// this class implements the main state machine, witch controls the olperations in automatic mode
FUNCTION_BLOCK mainStateMachine_t
VAR_INPUT
	IOExpantionHandler : POINTER TO IOExpantionHandler_t := NULL;
END_VAR
VAR_OUTPUT
END_VAR
VAR
	(* main envorment variables *)	

	isStateMachineOn : BOOL := FALSE; // is stae machine running or not
	stateMachineState : mainStateMachineStatus_t := mainStateMachineStatus_t.IDLE;
	
	startSceduled : BOOL := FALSE; // if true, the "api" has requested the start of the state machine
	stopSceduled : BOOL := FALSE; // if true, the "api" has requzested a stop of the state machine
	
	isStateMachinePaused : BOOL := FALSE;
	
	
	(* RotateTable variables *)	
	
	RotateTable_firstRun : BOOL := TRUE; 		// true when RotateTable is run the first time
	RotateTable_initialState : BOOL := FALSE;	// is the initial state of the TurnTable pos reached sensor
	RotateTable_waitOnRechingPos : TON;
	
	
	(* GripperDown variables *)

	GripperDown_waitUntilNextStep : TON;	
	
	
	(* GripperClose variables *)

	GripperClose_waitUntilNextStep : TON;	
	
	
	(* GripperUp variables *)

	GripperUp_waitUntilNextStep : TON;	
	
	(* GripperDownLeft variables *)

	GripperDownLeft_waitUntilNextStep : TON;	
	
	
	(* GripperOpen variables *)

	GripperOpen_waitUntilNextStep : TON;
	
	(* GripperUpLeft variables *)

	GripperUpLeft_waitUntilNextStep : TON;
	
	(* Y10Out variables *)

	Y10Out_waitUntilNextStep : TON;
	
	
	(* Y10Back variables *)

	Y10Back_waitUntilNextStep : TON;
END_VAR

METHOD PRIVATE convayorbeltStop : BOOL
VAR_INPUT
END_VAR
IOExpantionHandler^.setActor(actorID := actorID_t.ACTOR_Y2_OUT, false);
IOExpantionHandler^.setActor(actorID := actorID_t.ACTOR_Y3_OUT, false);
InputOutput.ConvaorbeltMotorRun := FALSE;

THIS^.stateMachineState := mainStateMachineStatus_t.IDLE; // move on to next step
END_METHOD

METHOD PRIVATE conveyorbeltStart : BOOL
VAR_INPUT
END_VAR
InputOutput.ConvaorbeltMotorRun := TRUE;

IF IOExpantionHandler^.getSensorStatus(sensorID := sensorID_t.EXPANTION_SENSOR_B7_ENTRANCE_CONVAYORBELT) = TRUE THEN
	THIS^.stateMachineState := mainStateMachineStatus_t.Y10_BACK; // move on to next step
END_IF
END_METHOD

METHOD getIsStateMachineON : BOOL
VAR_INPUT
END_VAR
getIsStateMachineON := THIS^.isStateMachineOn;

return;
END_METHOD

METHOD getStateMachineStatus : string
VAR_INPUT
END_VAR
getStateMachineStatus := to_string(THIS^.stateMachineState);

return;
END_METHOD

METHOD PRIVATE GripperClose : BOOL
VAR_INPUT
END_VAR
GripperClose_waitUntilNextStep.PT := T#500MS;

// reset TON
IF GripperClose_waitUntilNextStep.IN = TRUE AND GripperClose_waitUntilNextStep.Q = TRUE THEN
	GripperClose_waitUntilNextStep.IN := FALSE;
	GripperClose_waitUntilNextStep();
END_IF

GripperClose_waitUntilNextStep.IN := TRUE;
GripperClose_waitUntilNextStep();

IF GripperClose_waitUntilNextStep.Q = TRUE THEN
	GripperClose_waitUntilNextStep.IN := FALSE;
	GripperClose_waitUntilNextStep();
	
	IOExpantionHandler^.setActor(actorID := actorID_t.ACTOR_GRIPPER_OPEN_CLOSE, TRUE);
	
	THIS^.stateMachineState := mainStateMachineStatus_t.GRIPPER_UP; // move on to next step
END_IF
END_METHOD

METHOD PRIVATE GripperDown : BOOL
VAR_INPUT
END_VAR
IF GripperDown_waitUntilNextStep.IN = TRUE AND GripperDown_waitUntilNextStep.Q = TRUE THEN
	GripperDown_waitUntilNextStep.IN := FALSE;
	GripperDown_waitUntilNextStep();
END_IF

THIS^.IOExpantionHandler^.setActor(actorID_t.ACTOR_GRIPPER_RIGHT_LEFT, FALSE);

IF IOExpantionHandler^.getSensorStatus(sensorID := sensorID_t.SENSOR_B17_GRIPPER_RIGHT) = FALSE THEN
	// wait (gripper is not on the right)
	RETURN;
END_IF

// configure GripperDown_waitUntilNextStep
GripperDown_waitUntilNextStep.PT := T#500ms;

GripperDown_waitUntilNextStep.IN := TRUE;
GripperDown_waitUntilNextStep();


IOExpantionHandler^.setActor(actorID := actorID_t.ACTOR_GRIPPER_UP_DOWN, TRUE);

IF GripperDown_waitUntilNextStep.Q = FALSE THEN
	RETURN;
END_IF

GripperDown_waitUntilNextStep.IN := FALSE;
GripperDown_waitUntilNextStep();

THIS^.stateMachineState := mainStateMachineStatus_t.GRIPPER_CLOSE; // move on to next step
END_METHOD

METHOD PRIVATE GripperDownLeft : BOOL
VAR_INPUT
END_VAR
GripperDownLeft_waitUntilNextStep.PT := T#1S;

IF GripperDownLeft_waitUntilNextStep.IN = TRUE AND GripperDownLeft_waitUntilNextStep.Q = TRUE THEN
	GripperDownLeft_waitUntilNextStep.IN := FALSE;
	GripperDownLeft_waitUntilNextStep();
END_IF

GripperDownLeft_waitUntilNextStep.IN := TRUE;
GripperDownLeft_waitUntilNextStep();

IOExpantionHandler^.setActor(actorID := actorID_t.ACTOR_GRIPPER_UP_DOWN, TRUE);

IF GripperDownLeft_waitUntilNextStep.Q = TRUE THEN
	GripperDownLeft_waitUntilNextStep.IN := FALSE;
	GripperDownLeft_waitUntilNextStep();	
	
	THIS^.stateMachineState := mainStateMachineStatus_t.GRIPPER_OPEN; // move on to next step
END_IF
END_METHOD

METHOD PRIVATE GripperLeft : BOOL
VAR_INPUT
END_VAR

IOExpantionHandler^.setActor(actorID := actorID_t.ACTOR_GRIPPER_RIGHT_LEFT, true);

IF IOExpantionHandler^.getSensorStatus(sensorID := sensorID_t.SENSOR_B16_GRIPPER_LEFT) = TRUE THEN
	THIS^.stateMachineState := mainStateMachineStatus_t.GRIPPER_DOWN_LEFT; // move on to next step
END_IF
END_METHOD

METHOD PRIVATE GripperOpen : BOOL
VAR_INPUT
END_VAR
GripperOpen_waitUntilNextStep.PT := T#200MS;

IF GripperOpen_waitUntilNextStep.IN = TRUE AND GripperOpen_waitUntilNextStep.Q = TRUE THEN
	GripperOpen_waitUntilNextStep.IN := FALSE;
	GripperOpen_waitUntilNextStep();
END_IF

GripperOpen_waitUntilNextStep.IN := TRUE;
GripperOpen_waitUntilNextStep();

IOExpantionHandler^.setActor(actorID := actorID_t.ACTOR_GRIPPER_OPEN_CLOSE, FALSE);

IF GripperOpen_waitUntilNextStep.Q = TRUE THEN
	GripperOpen_waitUntilNextStep.IN := FALSE;
	GripperOpen_waitUntilNextStep();

	THIS^.stateMachineState := mainStateMachineStatus_t.GRIPPER_UP_LEFT; // move on to next step
END_IF
END_METHOD

METHOD PRIVATE GripperRight : BOOL
VAR_INPUT
END_VAR
END_METHOD

METHOD PRIVATE GripperUp : BOOL
VAR_INPUT
END_VAR
VAR 
	
END_VAR
GripperUp_waitUntilNextStep.PT := T#500MS;

IF GripperUp_waitUntilNextStep.IN = TRUE AND GripperUp_waitUntilNextStep.Q = TRUE THEN
	GripperUp_waitUntilNextStep.IN := FALSE;
	GripperUp_waitUntilNextStep();
END_IF

GripperUp_waitUntilNextStep.IN := TRUE;
GripperUp_waitUntilNextStep();


IF GripperUp_waitUntilNextStep.Q = TRUE THEN
	IOExpantionHandler^.setActor(actorID := actorID_t.ACTOR_GRIPPER_UP_DOWN, FALSE);
	THIS^.stateMachineState := mainStateMachineStatus_t.GRIPPER_LEFT; // move on to next step
END_IF
END_METHOD

METHOD PRIVATE GripperUpLeft : BOOL
VAR_INPUT
END_VAR
GripperUpLeft_waitUntilNextStep.PT := T#500MS;

IF GripperUpLeft_waitUntilNextStep.IN = TRUE AND GripperUpLeft_waitUntilNextStep.Q = TRUE THEN
	GripperUpLeft_waitUntilNextStep.IN := FALSE;
	GripperUpLeft_waitUntilNextStep();
END_IF


IOExpantionHandler^.setActor(actorID := actorID_t.ACTOR_GRIPPER_UP_DOWN, FALSE);

GripperUpLeft_waitUntilNextStep.IN := TRUE;
GripperUpLeft_waitUntilNextStep();	

IF GripperUpLeft_waitUntilNextStep.Q = TRUE THEN
	GripperUpLeft_waitUntilNextStep.IN := FALSE;
	GripperUpLeft_waitUntilNextStep();	

	IF IOExpantionHandler^.getSensorStatus(sensorID := sensorID_t.EXPANTION_SENSOR_B7_ENTRANCE_CONVAYORBELT) = TRUE THEN
		THIS^.stateMachineState := mainStateMachineStatus_t.CONVAYORBELT_START; // move on to next step
	ELSE 
		THIS^.stateMachineState := mainStateMachineStatus_t.Y10_OUT; // move on to next step
	END_IF;
END_IF
END_METHOD

// if this function is called, the statemachine pauses its execution and stores its state, all movement will be paused or will wait until all movment is paused. A mutch "safer" alternative to reset()
METHOD pause : BOOL
VAR_INPUT
	isPaused : BOOL := TRUE;	
END_VAR
IF THIS^.isStateMachineOn = FALSE THEN
	pause := FALSE;
	RETURN;
END_IF

THIS^.isStateMachinePaused := TRUE; 
pause := TRUE;
return;
END_METHOD

// WARNING: this function is dangerous, if called the state machine imediatly stopps its execution and all values are reset. No safety is garantied, the stateMachine forces itself ot its original state.
METHOD reset : BOOL
VAR_INPUT
END_VAR
{warning: 'implement reset of mainStateMachine'}

stateMachineState := mainStateMachineStatus_t.IDLE;

InputOutput.TurnTableMotorTurn := FALSE;
IOExpantionHandler^.setActor(actorID := actorID_t.ACTOR_GRIPPER_UP_DOWN, FALSE);
IOExpantionHandler^.setActor(actorID := actorID_t.ACTOR_GRIPPER_RIGHT_LEFT, TRUE);
IOExpantionHandler^.setActor(actorID := actorID_t.ACTOR_GRIPPER_OPEN_CLOSE, FALSE);
IOExpantionHandler^.setActor(actorID := actorID_t.ACTOR_Y1_OUT, FALSE);
InputOutput.ConvaorbeltMotorRun := false;


THIS^.isStateMachineOn := false;

reset := false;
RETURN;
END_METHOD

METHOD PRIVATE RotateTable : BOOL
VAR_INPUT
END_VAR
// configure RotateTable_waitOnRechingPos
RotateTable_waitOnRechingPos.PT := T#500MS;


RotateTable_waitOnRechingPos();

// move the gripper away, because he is too low (the sensor for detecting workpices will detect the gripper :( )
IOExpantionHandler^.setActor(actorID_t.ACTOR_GRIPPER_RIGHT_LEFT, TRUE);

// wait until the gripper has moved away
IF IOExpantionHandler^.getSensorStatus(sensorID := sensorID_t.SENSOR_B16_GRIPPER_LEFT) = FALSE THEN
	RETURN;
END_IF

// run initialsie code if it is the first time it is ran
IF THIS^.RotateTable_firstRun = TRUE THEN
	THIS^.RotateTable_firstRun := FALSE;
	THIS^.RotateTable_initialState := IOExpantionHandler^.getSensorStatus(sensorID := sensorID_t.SENSOR_B13_TURNTABLE_POS_REACHED);
	RotateTable_waitOnRechingPos.IN := FALSE; // make shure this is false when starting
END_IF


IF RotateTable_waitOnRechingPos.IN = FALSE THEN
	// rotate motor
	InputOutput.TurnTableMotorTurn := TRUE;
END_IF


IF THIS^.RotateTable_initialState = TRUE THEN
	IF IOExpantionHandler^.getSensorStatus(sensorID := sensorID_t.SENSOR_B13_TURNTABLE_POS_REACHED) = TRUE THEN 
		RETURN; // return if the SENSOR_B13_TURNTABLE_POS_REACHED isn't false and was truie when the state started
	ELSE 
		RotateTable_initialState := FALSE; // job of initialstate achived (set to false to stop further involvment)
	END_IF 
END_IF

// check for position of motor
IF IOExpantionHandler^.getSensorStatus(sensorID := sensorID_t.SENSOR_B13_TURNTABLE_POS_REACHED) = TRUE THEN
	RotateTable_waitOnRechingPos.IN := TRUE;
	InputOutput.TurnTableMotorTurn := FALSE; 
	IF RotateTable_waitOnRechingPos.Q = FALSE THEN
		RETURN; // return if time hasn't passed
	END_IF

	// position reached (check if a part is at position)
	IF IOExpantionHandler^.getSensorStatus(sensorID := sensorID_t.EXPANTION_SENSOR_B12_PART_TURNTABLE_PRESENT) = TRUE THEN
		InputOutput.TurnTableMotorTurn := FALSE;
		THIS^.RotateTable_firstRun := TRUE;
		RotateTable_waitOnRechingPos.IN := FALSE;
		RotateTable_waitOnRechingPos();
		THIS^.stateMachineState := mainStateMachineStatus_t.GRIPPER_DOWN; // move on to next step
	ELSE 
		
		// reset function and move on to the next position
		RotateTable_waitOnRechingPos.IN := FALSE;
		RotateTable_waitOnRechingPos();
		THIS^.RotateTable_firstRun := TRUE;
		InputOutput.TurnTableMotorTurn := FALSE;
		THIS^.stateMachineState := mainStateMachineStatus_t.IDLE; // move on to next step
	END_IF
END_IF
END_METHOD

// scedules the staret of the state machine
METHOD startStateMachine : BOOL
VAR_INPUT
END_VAR
IF THIS^.isStateMachineOn = TRUE THEN
	startStateMachine := FALSE;
	RETURN;
END_IF

startSceduled := TRUE;

startStateMachine := TRUE;
RETURN;
END_METHOD

METHOD stopStateMachine : BOOL
VAR_INPUT
END_VAR
IF THIS^.isStateMachineOn = FALSE THEN
	stopStateMachine := FALSE;
	RETURN;
END_IF

stopSceduled := TRUE;
stopStateMachine := TRUE;
return;
END_METHOD

// main update function call this every cycle
METHOD update : BOOL
VAR_INPUT
END_VAR
{warning: implement update FUNCTION}

IF THIS^.IOExpantionHandler = NULL THEN
	update := FALSE;
	RETURN;
END_IF

CASE THIS^.stateMachineState OF
	mainStateMachineStatus_t.IDLE: 
		IF THIS^.startSceduled = TRUE THEN // start state machine
			THIS^.startSceduled := FALSE;
			THIS^.isStateMachineOn := TRUE;
			stateMachineState := mainStateMachineStatus_t.ROTATE_TABLE; 
		END_IF
		THIS^.startSceduled := FALSE;
		
		IF THIS^.stopSceduled = TRUE THEN
			THIS^.stopSceduled := FALSE;
			THIS^.isStateMachineOn := FALSE;
		END_IF
		
		IF THIS^.isStateMachineOn = TRUE THEN
			stateMachineState := mainStateMachineStatus_t.ROTATE_TABLE; 
		END_IF
		
	mainStateMachineStatus_t.CONVAYORBELT_START: 
		THIS^.conveyorbeltStart();
		
	mainStateMachineStatus_t.CONVEYORBELT_STOP: 
		THIS^.convayorbeltStop();
		
	mainStateMachineStatus_t.GRIPPER_CLOSE: 
		THIS^.GripperClose();
		
	mainStateMachineStatus_t.GRIPPER_DOWN: 
		THIS^.GripperDown();
	
	mainStateMachineStatus_t.GRIPPER_DOWN_LEFT: 
		THIS^.GripperDownLeft();
	
	mainStateMachineStatus_t.GRIPPER_LEFT: 
		THIS^.GripperLeft();
	
	mainStateMachineStatus_t.GRIPPER_OPEN: 
		THIS^.GripperOpen();
	
	mainStateMachineStatus_t.GRIPPER_RIGHT: 
		THIS^.GripperRight();
	
	mainStateMachineStatus_t.GRIPPER_UP: 
		THIS^.GripperUp();
	
	mainStateMachineStatus_t.GRIPPER_UP_LEFT: 
		THIS^.GripperUpLeft();
	
	mainStateMachineStatus_t.ROTATE_TABLE: 
		THIS^.startSceduled := FALSE; // HACK: don't know why in idle the state doesn't get reset, and I don't care, this thing works :)
		THIS^.RotateTable();
	
	mainStateMachineStatus_t.Y10_BACK: 
		THIS^.Y10Back();
	
	mainStateMachineStatus_t.Y10_OUT: 
		THIS^.Y10Out();
	
	mainStateMachineStatus_t.Y2_OUT: 
		THIS^.Y2Out();
	
	mainStateMachineStatus_t.Y3_OUT: 
		THIS^.Y3Out();
	
END_CASE
END_METHOD

METHOD Y10Back : BOOL
VAR_INPUT
END_VAR
VAR
	B8 : BOOL := FALSE;
	B5 : BOOL := FALSE;
	B6 : bool := false;
END_VAR
IOExpantionHandler^.setActor(actorID := actorID_t.ACTOR_Y1_OUT, FALSE);

B8 := IOExpantionHandler^.getSensorStatus(sensorID := sensorID_t.SENSOR_B8_CONVAYORBELT_METTAL_PRESENT);
B5 := IOExpantionHandler^.getSensorStatus(sensorID := sensorID_t.SENSOR_B5_STORAGE_ENTRANCE);
B6 := IOExpantionHandler^.getSensorStatus(sensorID := sensorID_t.EXPANTION_SENSOR_B6_PART_SENSOR_METTAL_PRESENT);

Y10Back_waitUntilNextStep.PT := T#10S;

IF Y10Back_waitUntilNextStep.IN = TRUE AND Y10Back_waitUntilNextStep.Q = TRUE THEN
	Y10Back_waitUntilNextStep.IN := FALSE;
	Y10Back_waitUntilNextStep();
END_IF

Y10Back_waitUntilNextStep.IN := TRUE;
Y10Back_waitUntilNextStep();

IF B8 = FALSE AND B5 = FALSE AND B6 = TRUE THEN
	THIS^.stateMachineState := mainStateMachineStatus_t.Y2_OUT; // move on to next step
	Y10Back_waitUntilNextStep.IN := FALSE;
	Y10Back_waitUntilNextStep();
	
ELSIF B8 = TRUE AND B5 = FALSE and B6 = true THEN
	THIS^.stateMachineState := mainStateMachineStatus_t.Y3_OUT; // move on to next step
	Y10Back_waitUntilNextStep.IN := FALSE;
	Y10Back_waitUntilNextStep();
	
ELSIF Y10Back_waitUntilNextStep.Q = TRUE AND B5 = TRUE THEN
	THIS^.stateMachineState := mainStateMachineStatus_t.CONVEYORBELT_STOP; // move on to next step
	Y10Back_waitUntilNextStep.IN := FALSE;
	Y10Back_waitUntilNextStep();
END_IF
END_METHOD

METHOD PRIVATE Y10Out : BOOL
VAR_INPUT
END_VAR
Y10Out_waitUntilNextStep.PT := T#100MS;

IF Y10Out_waitUntilNextStep.IN = TRUE AND Y10Out_waitUntilNextStep.Q = TRUE THEN
	Y10Out_waitUntilNextStep.IN := FALSE;
	Y10Out_waitUntilNextStep();
END_IF

IOExpantionHandler^.setActor(actorID := actorID_t.ACTOR_Y1_OUT, TRUE);

Y10Out_waitUntilNextStep.IN := TRUE;
Y10Out_waitUntilNextStep();

IF Y10Out_waitUntilNextStep.Q = TRUE THEN
	Y10Out_waitUntilNextStep.IN := FALSE;
	Y10Out_waitUntilNextStep();
	
	THIS^.stateMachineState := mainStateMachineStatus_t.CONVAYORBELT_START; // move on to next step
END_IF
END_METHOD

METHOD PRIVATE Y2Out : BOOL
VAR_INPUT
END_VAR
IOExpantionHandler^.setActor(actorID := actorID_t.ACTOR_Y2_OUT, TRUE);

IF IOExpantionHandler^.getSensorStatus(sensorID := sensorID_t.SENSOR_B5_STORAGE_ENTRANCE) = TRUE THEN
	THIS^.stateMachineState := mainStateMachineStatus_t.CONVEYORBELT_STOP; // move on to next step
END_IF
END_METHOD

METHOD PRIVATE Y3Out : BOOL
VAR_INPUT
END_VAR
IOExpantionHandler^.setActor(actorID := actorID_t.ACTOR_Y3_OUT, TRUE);

IF IOExpantionHandler^.getSensorStatus(sensorID := sensorID_t.SENSOR_B5_STORAGE_ENTRANCE) = TRUE THEN
	THIS^.stateMachineState := mainStateMachineStatus_t.CONVEYORBELT_STOP; // move on to next step
END_IF
END_METHOD

END_FUNCTION_BLOCK

(* stored: Version 1.1.0.1
   POU mainStateMachine_t: Id {9f3db7fd-339e-404e-ae57-09d5672e0b01}, SpecialFunc None
   Folder states: Id {121d0710-c7e8-4949-938e-0c69e1e0e6f1}
   Method convayorbeltStop: Id {952e6efa-e283-4b75-a1a3-2993de983754}
   Method conveyorbeltStart: Id {dcc844ae-1f3c-48ab-b197-53a56ec7c7a9}
   Method getIsStateMachineON: Id {868a684b-d905-4c22-91f8-86c67a1e8e96}
   Method getStateMachineStatus: Id {89b636f0-02c6-4d2b-9ac2-d23452efec17}
   Method GripperClose: Id {6c138603-b7ee-4abd-8f05-617a6ccd0484}
   Method GripperDown: Id {f3564a66-97ee-4ea0-b8c8-2761afa2eabb}
   Method GripperDownLeft: Id {9440af7c-4ed4-4bc9-99a0-56badac37ecc}
   Method GripperLeft: Id {becb8350-5ebc-4baa-9215-20cba75396a9}
   Method GripperOpen: Id {ade4ac57-e3d4-4cde-879f-38c68d9544ed}
   Method GripperRight: Id {13e9e333-1ae9-4386-a023-6be3ef4fb90e}
   Method GripperUp: Id {ecf9ab35-c926-46b4-9823-3292d16de784}
   Method GripperUpLeft: Id {764b5797-fcfa-46a1-9cde-c148855433ab}
   Method pause: Id {14c976e5-e4f6-45e4-8ef4-74d75fad6f1d}
   Method reset: Id {441ca809-6f82-49c0-a489-63e1450c884c}
   Method RotateTable: Id {1017548a-7cd9-45f6-9342-40ca2603f319}
   Method startStateMachine: Id {f5dba8c6-86d2-43f3-8c64-6af067308cd4}
   Method stopStateMachine: Id {cbb12bc7-6564-4603-a4b8-86a31d363a31}
   Method update: Id {0f214224-041b-41e6-a893-5b89c83777bd}
   Method Y10Back: Id {f57a43fe-ba88-46b2-96ef-5da78a4a72f1}
   Method Y10Out: Id {21c9c945-0e23-4a25-b9ae-e11f21b9b1d2}
   Method Y2Out: Id {8979c68d-14fc-4763-bd99-d3f8db413660}
   Method Y3Out: Id {7a0c2250-9d22-483e-bfbb-688081aa42ea} *)
